(*
    CLI fixture. A suite that EXTENDS the user-defined intermediate base
    FB_TestSuiteWithClock through a library-qualified spelling, the way real
    TcUnit-flavored source names it.
*)
FUNCTION_BLOCK FB_ClockAdvancingSuiteTests EXTENDS TcUnit.FB_TestSuiteWithClock

AdvancesPastTimeout();

METHOD PRIVATE AdvancesPastTimeout
TEST('AdvancesPastTimeout');

AdvanceClockMs(Duration := T#500MS);

AssertTrue(Condition := TRUE,
           Message := 'suite reachable through the qualified EXTENDS chain');

TEST_FINISHED();
END_METHOD

END_FUNCTION_BLOCK

(* stored: Version 1.1.0.1, ProductVersion 3.1.4026.18
   POU FB_ClockAdvancingSuiteTests: Id {267d7f54-cead-459f-9b43-6ee4e810c1a2}, SpecialFunc None
   Method AdvancesPastTimeout: Id {267d7f54-cead-459f-9b43-6ee4e810c1a3} *)
